// TwinCAT 3 PLC project TCPServer
// ProgramVersion: 3.1.4022.7
// libraries:
//   Tc2_Standard, * (Beckhoff Automation GmbH)
//   Tc2_System, * (Beckhoff Automation GmbH)
//   Tc2_TcpIp, * (Beckhoff Automation GmbH)
//   Tc3_Module, * (Beckhoff Automation GmbH)
// project tree:
//   / PlcTask.TcTTO (not stored)
//   POUs/ FB_TCPServer.TcPOU, MAIN.TcPOU
// real-time tasks:
//   TASK PlcTask: cycle T#10ms, priority 20, ADS port 350

// ---- POUs/FB_TCPServer.TcPOU
FUNCTION_BLOCK FB_TCPServer
VAR_INPUT
	sLocalHost: T_IPv4Addr;
	nLocalPort: UDINT;
	bStartCommunication : BOOL;
END_VAR
VAR_OUTPUT
	bConnected: BOOL;
	sSendData: STRING(255);
	arrSendData: ARRAY[0..3] OF BYTE;
	bBusy: BOOL;	
	bError: BOOL;
	nErrorID: UDINT;
END_VAR
VAR
	iState: INT;
	hListener: T_HSOCKET;
	hSocket: T_HSOCKET;
	fbSocketAccept: FB_SocketAccept;
	fbSocketListen: FB_SocketListen;
	fbSocketReceive: FB_SocketReceive;
	fbSocketClose: FB_SocketClose;
	fbSocketCloseAll: FB_SocketCloseAll;
	fbSocketSend: FB_SocketSend;
	bAcceptExecute: BOOL;
	
	ReceiveCounter: UDINT;
	nSocketSendErrorID: UDINT;
	sReadData: STRING(255);
	arrReadData: ARRAY[0..3] OF BYTE;
	received_value: UDINT; 
	nRecBytes: UDINT; 
	
	bSendTrigger: BOOL;
END_VAR

CASE iState OF
0: // Init State
	IF bStartCommunication = TRUE  THEN
		fbSocketListen(bExecute := FALSE);
		fbSocketAccept(bExecute := FALSE);
		fbSocketCloseAll(bExecute := FALSE);
		fbSocketClose(bExecute:= FALSE);
		bBusy := TRUE;
		iState := iState + 10;
	ELSE
		bBusy := FALSE;
	END_IF
	
10:
	fbSocketListen(																// Open Listener-Socket
		sSrvNetId:= '', 														// Local NetID
		sLocalHost:= sLocalHost, 												// Local IP
		nLocalPort:= nLocalPort, 												// Local Port
		bExecute:= TRUE, 
		tTimeout:= T#4S, 
		bBusy=> , 
		bError=> bError, 
		nErrId=> nErrorID,
		hListener=> hListener);													// Handle of Listener Socket
		
	IF hListener.handle <> 0 THEN
		iState := iState + 10;	
	ELSIF bError THEN
		iState := 40;
	END_IF
	
20: 		
	fbSocketAccept(																// Accept Client connection
		sSrvNetId:= '', 		
		hListener:= hListener, 													// Handle of Listener Socket
		bExecute:= TRUE, 
		tTimeout:= T#4S, 
		bAccepted=> , 
		bBusy=> , 
		bError=> bError, 
		nErrId=> nErrorID,
		hSocket=> hSocket);														// Connection Handle
	IF NOT fbSocketAccept.bBusy THEN
		fbSocketAccept(bExecute:= FALSE);
	END_IF

	IF bError THEN
		iState := 40; 
	ELSIF hSocket.handle <> 0 THEN
		iState := iState + 10; 
		bConnected := TRUE;
	END_IF
	
30: // Receive Data
	fbSocketReceive(															// Check cyclically for new client telegrams 
		sSrvNetId:= '', 
		hSocket:= hSocket, 
		cbLen:= SIZEOF(arrReadData) , 
		pDest:= ADR(arrReadData), 
		bExecute:= TRUE, 														
		tTimeout:= T#300S, 
		bBusy=> , 
		bError=> bError, 
		nErrId=> nErrorID,
		nRecBytes=> nRecBytes);
		
	IF nRecBytes = 4 THEN  
    // Copy the received bytes  
    received_value := (DWORD_TO_UDINT(arrReadData[0]) * 16777216) + (DWORD_TO_UDINT(arrReadData[1]) * 65536) +  
                      (DWORD_TO_UDINT(arrReadData[2]) * 256) + DWORD_TO_UDINT(arrReadData[3]);  
	END_IF  
		
	IF NOT fbSocketReceive.bBusy THEN
		fbSocketReceive(bExecute := FALSE);
		IF fbSocketReceive.nRecBytes <> 0 THEN									// Switch to send-state when data are received
			fbSocketSend(bExecute:= FALSE);
			ReceiveCounter := ReceiveCounter + 1; 
			memcpy(ADR(arrSendData), ADR(arrReadData), fbSocketReceive.nRecBytes);	// Copy received data from ReceiveBuffer to SendBuffer
			//memset(ADR(arrReadData), 0, SIZEOF(arrReadData));						// Empty ReceiveBuffer
			iState := iState + 5;
		END_IF
	END_IF
	IF fbSocketReceive.bError OR(NOT bStartCommunication) THEN					// Close connection when error is occuring or trigger is set
		iState := iState + 10;
	END_IF

35: // Send Data
	fbSocketSend(																// Send Data to client
		sSrvNetId:= '', 
		hSocket:= hSocket, 
		cbLen:= SIZEOF(arrSendData), 
		pSrc:= ADR(arrSendData),
		bExecute:= TRUE, 
		tTimeout:= T#20S, 
		bBusy=> , 
		bError=> bError, 
		nErrId=> nErrorID);	
	IF NOT fbSocketSend.bBusy THEN												// Switch back to receiving state after sending
		iState := iState - 5;
	ELSIF fbSocketSend.bError THEN
		nSocketSendErrorID := nErrorID;
		iState := iState + 5;													// Close connection in case of error 
	END_IF
	
40:	// Error Handling	
	fbSocketClose(																// Close Listener-Socket
		sSrvNetId:= '', 
		hSocket:= hListener, 
		bExecute:= TRUE, 
		tTimeout:= T#4S, 
		bBusy=> , 
		bError=> bError, 
		nErrId=> nErrorID);		
	IF (NOT fbSocketClose.bBusy) OR fbSocketClose.bError THEN
		hListener.handle := 0;
		iState := iState + 1;
	END_IF
41:	
	fbSocketClose(bExecute := FALSE);
	iState := iState + 1;
42:
	fbSocketClose(																// Close Connection Socket
		sSrvNetId:= '', 
		hSocket:= hSocket, 
		bExecute:= TRUE, 
		tTimeout:= T#4S, 
		bBusy=> , 
		bError=> bError, 
		nErrId=> nErrorID);
	IF NOT (fbSocketClose.bBusy) OR fbSocketClose.bError THEN
		hSocket.handle := 0;	
		iState := 0;
		bConnected := FALSE;
	END_IF
END_CASE

END_FUNCTION_BLOCK

// ---- POUs/MAIN.TcPOU
PROGRAM MAIN
VAR
	bInit: BOOL := TRUE;
	fbSocketCloseAll: FB_SocketCloseAll; 
	bSocketCloseError: BOOL;
	nSocketCloseError: UDINT;	
	nServer1Port				: UDINT 				:= 5050;
	sServer1Host				: T_IPv4Addr 			:= '';		
		
	fbTcpEchoServer1				: FB_TCPServer;
		sServerReceivedData			: STRING(255);
		bStartServer1Communication	: BOOL 					:= TRUE;
		bServer1Connected			: BOOL;
		sServerData					: STRING(255);
		bServer1Busy				: BOOL;
		bServer1Error				: BOOL;
		nServer1ErrorID				: UDINT;
	
	bAutogenerateData				: BOOL 					:= TRUE;
	fbTimer1						: TON;
	nCnt							: UDINT;
END_VAR

IF bInit THEN 				// Init Step to close all sockets after login PLC with  downlaod
	fbSocketCloseAll(
		sSrvNetId:= '', 
		bExecute:= TRUE, 
		tTimeout:= T#3S, 
		bBusy=> , 
		bError=> bSocketCloseError, 
		nErrId=> nSocketCloseError);
	IF NOT (fbSocketCloseAll.bBusy OR fbSocketCloseAll.bError) THEN
		bInit := FALSE;
		fbSocketCloseAll(bExecute:= FALSE);
	END_IF
ELSE
		
	fbTcpEchoServer1(
		sLocalHost:= '192.168.17.110', 											// Server IP Adress
		nLocalPort:= nServer1Port, 									// Server port
		bStartCommunication:= bStartServer1Communication, 			// Allow Client-connection or close connection
		bConnected => bServer1Connected,							// Client connection is valid
		sSendData => sServerData,
		bBusy=> bServer1Busy, 
		bError=> bServer1Error, 
		nErrorID=> nServer1ErrorID);
END_IF

END_PROGRAM
